// Mitsubishi GX Works2 project: BookEX3_8 Device   PLC: Q13UDV

TYPE DateTime : STRUCT
  Year : INT;
  Month : INT;
  Day : INT;
  WeekDay : INT;
  iHour : INT;
  iMin : INT;
  iSec : INT;
  ms : INT;
END_STRUCT END_TYPE

TYPE Vector : STRUCT
  axisX : REAL;
  axisY : REAL;
  axisZ : REAL;
END_STRUCT END_TYPE

TYPE WordBit : STRUCT
  Data : DWORD;
  Flag : BOOL;
END_STRUCT END_TYPE

// global labels: Global
VAR_GLOBAL
  bVar0 AT M5000 : BOOL;
  abArray0 AT M5010 : ARRAY [0..49] OF BOOL;
  sStr0 AT D5000 : STRING[199];
  sStr1 AT D5100 : STRING[199];
  sStr2 AT D5200 : STRING[199];
  sStr3 AT D5300 : STRING[199];
  sStr4 AT D5400 : STRING[199];
  sStr5 AT D5500 : STRING[199];
  sStr6 AT D5600 : STRING[199];
  sStr7 AT D5700 : STRING[199];
  sStr8 AT D5800 : STRING[199];
  sStr9 AT D5900 : STRING[199];
  iVar0 AT D4500 : INT;
  iVar1 AT D4501 : INT;
  iVar2 AT D4502 : INT;
  iVar3 AT D4503 : INT;
  iVar4 AT D4504 : INT;
  iVar5 AT D4505 : INT;
  iVar6 AT D4506 : INT;
  iVar7 AT D4507 : INT;
  iVar8 AT D4508 : INT;
  iVar9 AT D4509 : INT;
  dVar0 AT D4510 : DINT;
  dVar1 AT D4512 : DINT;
  dVar2 AT D4514 : DINT;
  dVar3 AT D4516 : DINT;
  dVar4 AT D4518 : DINT;
  dVar5 AT D4520 : DINT;
  dVar6 AT D4522 : DINT;
  dVar7 AT D4524 : DINT;
  dVar8 AT D4526 : DINT;
  dVar9 AT D4528 : DINT;
  wVar0 AT D4530 : WORD;
  wVar1 AT D4531 : WORD;
  wVar2 AT D4532 : WORD;
  wVar3 AT D4533 : WORD;
  wVar4 AT D4534 : WORD;
  wVar5 AT D4535 : WORD;
  wVar6 AT D4536 : WORD;
  wVar7 AT D4537 : WORD;
  wVar8 AT D4538 : WORD;
  wVar9 AT D4539 : WORD;
  dwVar0 AT D4540 : DWORD;
  dwVar1 AT D4542 : DWORD;
  dwVar2 AT D4544 : DWORD;
  dwVar3 AT D4546 : DWORD;
  dwVar4 AT D4548 : DWORD;
  dwVar5 AT D4550 : DWORD;
  dwVar6 AT D4552 : DWORD;
  dwVar7 AT D4554 : DWORD;
  dwVar8 AT D4556 : DWORD;
  dwVar9 AT D4558 : DWORD;
  fsVar0 AT D4560 : REAL;
  fsVar1 AT D4562 : REAL;
  fsVar2 AT D4564 : REAL;
  fsVar3 AT D4566 : REAL;
  fsVar4 AT D4568 : REAL;
  fsVar5 AT D4570 : REAL;
  fsVar6 AT D4572 : REAL;
  fsVar7 AT D4574 : REAL;
  fsVar8 AT D4576 : REAL;
  fsVar9 AT D4578 : REAL;
  fdVar0 AT D4580 : LREAL;
  tTime0 AT D4620 : TIME;
  tTime1 AT D4622 : TIME;
  tTime2 AT D4624 : TIME;
  tTime3 AT D4626 : TIME;
  tTime4 AT D4628 : TIME;
  tTime5 AT D4630 : TIME;
  tTime6 AT D4632 : TIME;
  tTime7 AT D4634 : TIME;
  tTime8 AT D4636 : TIME;
  tTime9 AT D4638 : TIME;
  tTime10 AT D4640 : TIME;
  bVar1 AT M5001 : BOOL;
  bVar2 AT M5002 : BOOL;
  bVar3 AT M5003 : BOOL;
  bVar4 AT M5004 : BOOL;
  bVar5 AT M5005 : BOOL;
  bVar6 AT M5006 : BOOL;
  bVar7 AT M5007 : BOOL;
  bVar8 AT M5008 : BOOL;
  bVar9 AT M5009 : BOOL;
  abArray1 AT M5060 : ARRAY [0..49] OF BOOL;
  abArray2 AT M5110 : ARRAY [0..49] OF BOOL;
  abArray3 AT M5160 : ARRAY [0..49] OF BOOL;
  abArray4 AT M5210 : ARRAY [0..49] OF BOOL;
  abArray5 AT M5260 : ARRAY [0..49] OF BOOL;
  abArray6 AT M5310 : ARRAY [0..49] OF BOOL;
  abArray7 AT M5360 : ARRAY [0..49] OF BOOL;
  abArray8 AT M5410 : ARRAY [0..49] OF BOOL;
  abArray9 AT M5460 : ARRAY [0..49] OF BOOL;
  fdVar1 AT D4584 : LREAL;
  fdVar2 AT D4588 : LREAL;
  fdVar3 AT D4592 : LREAL;
  fdVar4 AT D4596 : LREAL;
  fdVar5 AT D4600 : LREAL;
  fdVar6 AT D4604 : LREAL;
  fdVar7 AT D4608 : LREAL;
  fdVar8 AT D4612 : LREAL;
  fdVar9 AT D4616 : LREAL;
  afsPen0 AT D2000 : ARRAY [0..499] OF REAL;
  afsPen1 AT D3000 : ARRAY [0..499] OF REAL;
END_VAR
// user libraries (not included): HMI

PROGRAM 000ConversionLD
VAR
  GetInt : INT;
  NthBit : INT;
  SetInt : INT;
  SetInt2 : INT;
END_VAR
(* structured ladder/FBD written out as ST: instructions are called as NAME(EN, inputs, outputs); _pN, _eN, _tN stand for wires *)
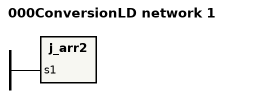
(* network 1 *)
(* element kind 9 j_arr2 <- TRUE *)
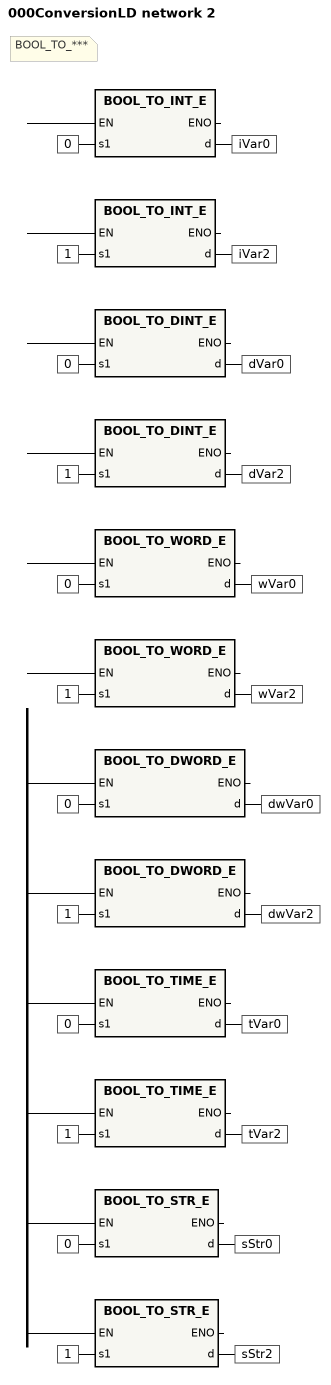
(* network 2 *)
(* BOOL_TO_*** *)
BOOL_TO_INT_E(TRUE, 0, iVar0);
BOOL_TO_INT_E(TRUE, 1, iVar2);
BOOL_TO_DINT_E(TRUE, 0, dVar0);
BOOL_TO_DINT_E(TRUE, 1, dVar2);
BOOL_TO_WORD_E(TRUE, 0, wVar0);
BOOL_TO_WORD_E(TRUE, 1, wVar2);
BOOL_TO_DWORD_E(TRUE, 0, dwVar0);
BOOL_TO_DWORD_E(TRUE, 1, dwVar2);
BOOL_TO_TIME_E(TRUE, 0, tVar0);
BOOL_TO_TIME_E(TRUE, 1, tVar2);
BOOL_TO_STR_E(TRUE, 0, sStr0);
BOOL_TO_STR_E(TRUE, 1, sStr2);
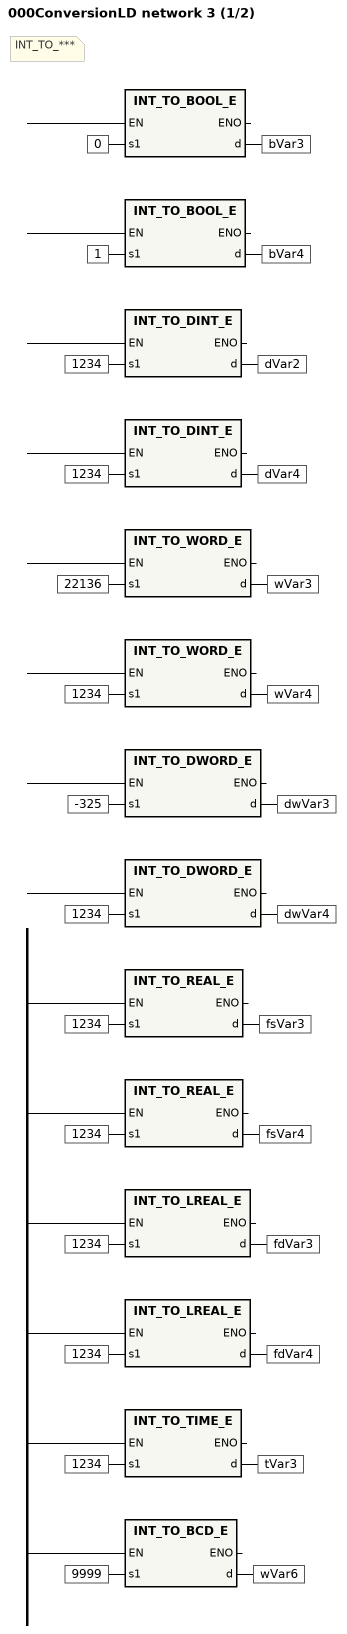
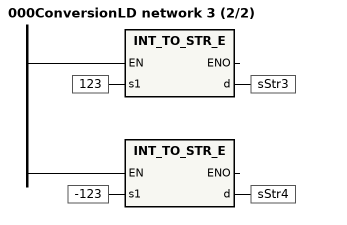
(* network 3 *)
(* INT_TO_*** *)
INT_TO_BOOL_E(TRUE, 0, bVar3);
INT_TO_BOOL_E(TRUE, 1, bVar4);
INT_TO_DINT_E(TRUE, 1234, dVar2);
INT_TO_DINT_E(TRUE, 1234, dVar4);
INT_TO_WORD_E(TRUE, 22136, wVar3);
INT_TO_WORD_E(TRUE, 1234, wVar4);
INT_TO_DWORD_E(TRUE, -325, dwVar3);
INT_TO_DWORD_E(TRUE, 1234, dwVar4);
INT_TO_REAL_E(TRUE, 1234, fsVar3);
INT_TO_REAL_E(TRUE, 1234, fsVar4);
INT_TO_LREAL_E(TRUE, 1234, fdVar3);
INT_TO_LREAL_E(TRUE, 1234, fdVar4);
INT_TO_TIME_E(TRUE, 1234, tVar3);
INT_TO_BCD_E(TRUE, 9999, wVar6);
INT_TO_STR_E(TRUE, 123, sStr3);
INT_TO_STR_E(TRUE, -123, sStr4);
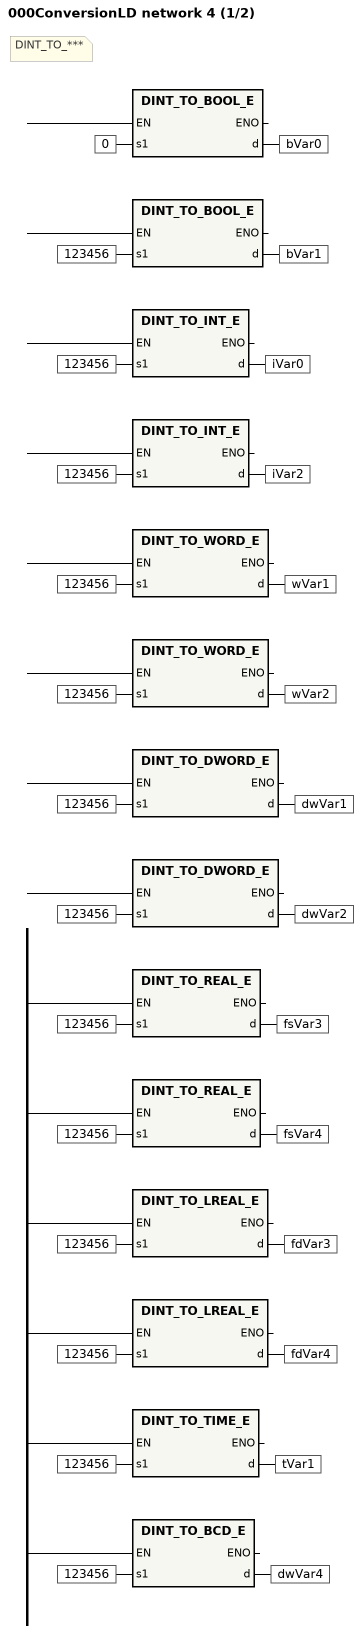
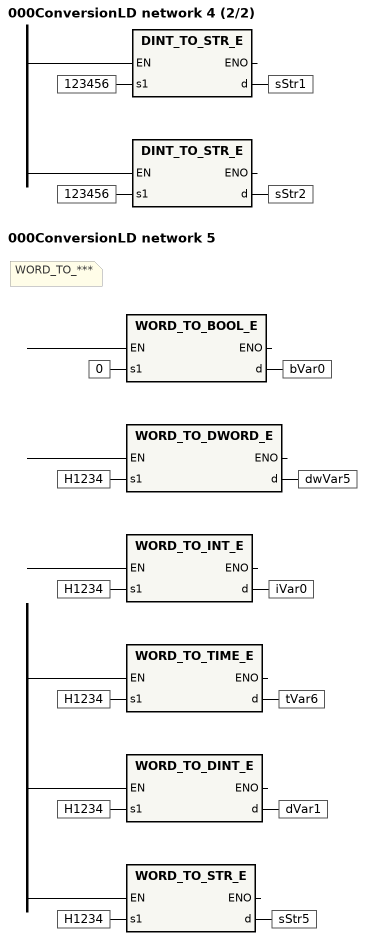
(* network 4 *)
(* DINT_TO_*** *)
DINT_TO_BOOL_E(TRUE, 0, bVar0);
DINT_TO_BOOL_E(TRUE, 123456, bVar1);
DINT_TO_INT_E(TRUE, 123456, iVar0);
DINT_TO_INT_E(TRUE, 123456, iVar2);
DINT_TO_WORD_E(TRUE, 123456, wVar1);
DINT_TO_WORD_E(TRUE, 123456, wVar2);
DINT_TO_DWORD_E(TRUE, 123456, dwVar1);
DINT_TO_DWORD_E(TRUE, 123456, dwVar2);
DINT_TO_REAL_E(TRUE, 123456, fsVar3);
DINT_TO_REAL_E(TRUE, 123456, fsVar4);
DINT_TO_LREAL_E(TRUE, 123456, fdVar3);
DINT_TO_LREAL_E(TRUE, 123456, fdVar4);
DINT_TO_TIME_E(TRUE, 123456, tVar1);
DINT_TO_BCD_E(TRUE, 123456, dwVar4);
DINT_TO_STR_E(TRUE, 123456, sStr1);
DINT_TO_STR_E(TRUE, 123456, sStr2);
(* network 5 *)
(* WORD_TO_*** *)
WORD_TO_BOOL_E(TRUE, 0, bVar0);
WORD_TO_DWORD_E(TRUE, H1234, dwVar5);
WORD_TO_INT_E(TRUE, H1234, iVar0);
WORD_TO_TIME_E(TRUE, H1234, tVar6);
WORD_TO_DINT_E(TRUE, H1234, dVar1);
WORD_TO_STR_E(TRUE, H1234, sStr5);
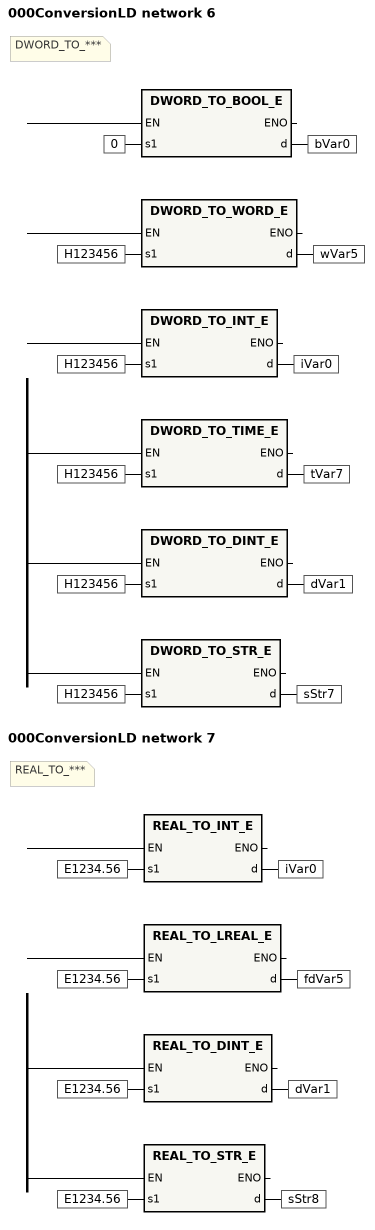
(* network 6 *)
(* DWORD_TO_*** *)
DWORD_TO_BOOL_E(TRUE, 0, bVar0);
DWORD_TO_WORD_E(TRUE, H123456, wVar5);
DWORD_TO_INT_E(TRUE, H123456, iVar0);
DWORD_TO_TIME_E(TRUE, H123456, tVar7);
DWORD_TO_DINT_E(TRUE, H123456, dVar1);
DWORD_TO_STR_E(TRUE, H123456, sStr7);
(* network 7 *)
(* REAL_TO_*** *)
REAL_TO_INT_E(TRUE, E1234.56, iVar0);
REAL_TO_LREAL_E(TRUE, E1234.56, fdVar5);
REAL_TO_DINT_E(TRUE, E1234.56, dVar1);
REAL_TO_STR_E(TRUE, E1234.56, sStr8);
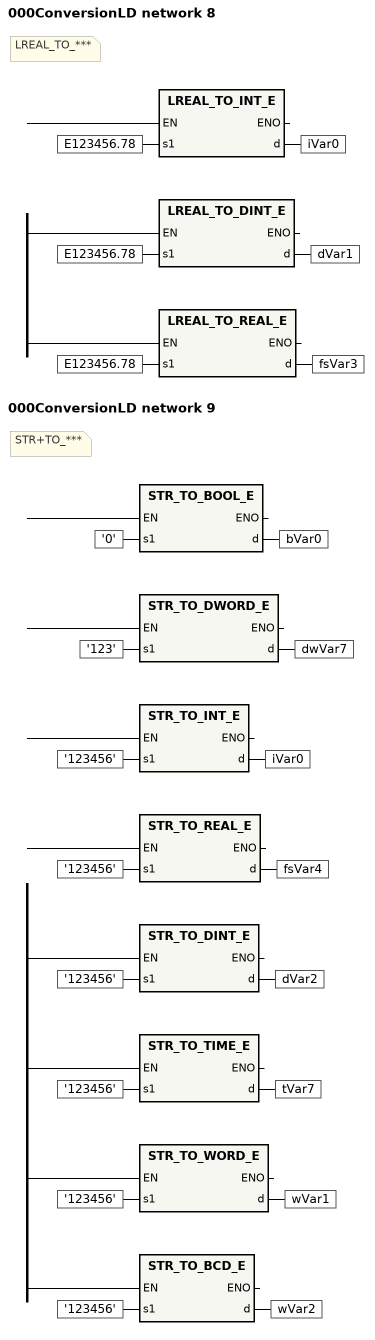
(* network 8 *)
(* LREAL_TO_*** *)
LREAL_TO_INT_E(TRUE, E123456.78, iVar0);
LREAL_TO_DINT_E(TRUE, E123456.78, dVar1);
LREAL_TO_REAL_E(TRUE, E123456.78, fsVar3);
(* network 9 *)
(* STR+TO_*** *)
STR_TO_BOOL_E(TRUE, '0', bVar0);
STR_TO_DWORD_E(TRUE, '123', dwVar7);
STR_TO_INT_E(TRUE, '123456', iVar0);
STR_TO_REAL_E(TRUE, '123456', fsVar4);
STR_TO_DINT_E(TRUE, '123456', dVar2);
STR_TO_TIME_E(TRUE, '123456', tVar7);
STR_TO_WORD_E(TRUE, '123456', wVar1);
STR_TO_BCD_E(TRUE, '123456', wVar2);
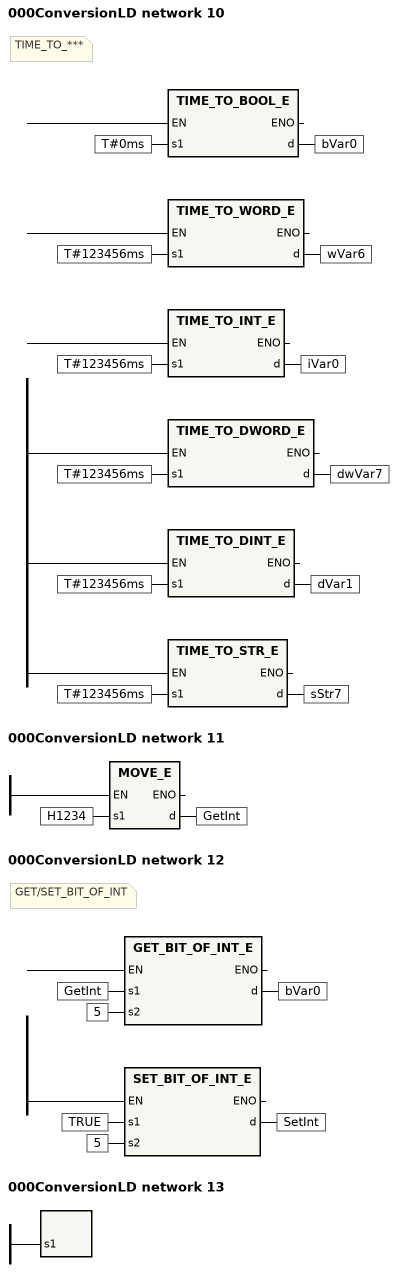
(* network 10 *)
(* TIME_TO_*** *)
TIME_TO_BOOL_E(TRUE, T#0ms, bVar0);
TIME_TO_WORD_E(TRUE, T#123456ms, wVar6);
TIME_TO_INT_E(TRUE, T#123456ms, iVar0);
TIME_TO_DWORD_E(TRUE, T#123456ms, dwVar7);
TIME_TO_DINT_E(TRUE, T#123456ms, dVar1);
TIME_TO_STR_E(TRUE, T#123456ms, sStr7);
(* network 11 Jmp11: *)
MOVE_E(TRUE, H1234, GetInt);
(* network 12 *)
(* GET/SET_BIT_OF_INT *)
GET_BIT_OF_INT_E(TRUE, GetInt, 5, bVar0);
SET_BIT_OF_INT_E(TRUE, TRUE, 5, SetInt);
(* network 13 *)
(* element kind 10  <- TRUE *)
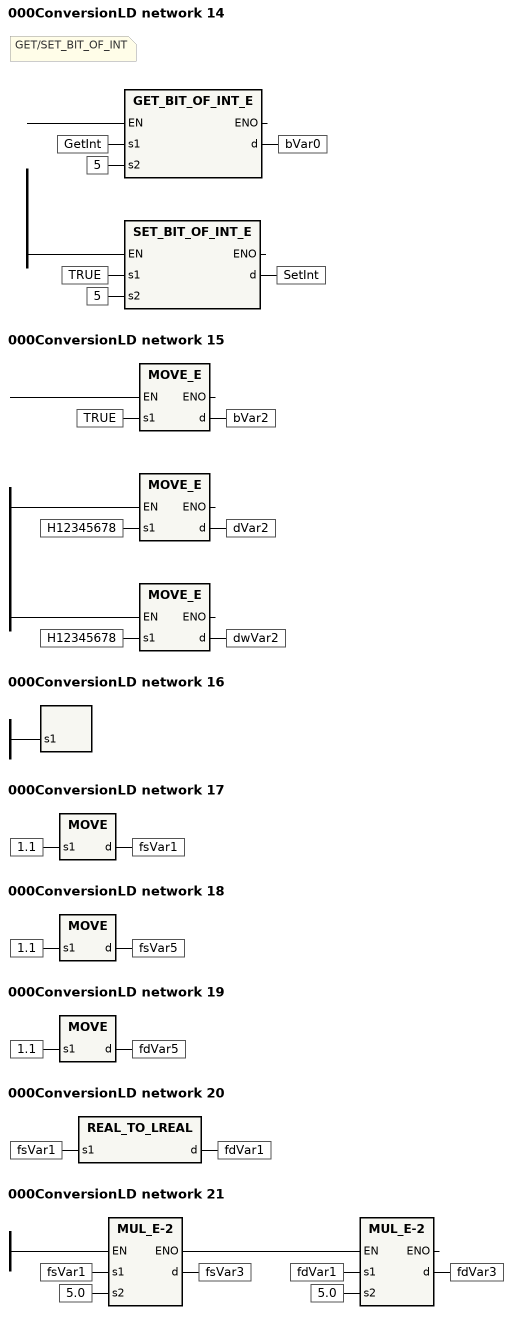
(* network 14 *)
(* GET/SET_BIT_OF_INT *)
GET_BIT_OF_INT_E(TRUE, GetInt, 5, bVar0);
SET_BIT_OF_INT_E(TRUE, TRUE, 5, SetInt);
(* network 15 Jmp15: *)
MOVE_E(TRUE, TRUE, bVar2);
MOVE_E(TRUE, H12345678, dVar2);
MOVE_E(TRUE, H12345678, dwVar2);
(* network 16 *)
(* element kind 10  <- TRUE *)
(* network 17 Jmp20: *)
fsVar1 := MOVE(1.1);
(* network 18 *)
fsVar5 := MOVE(1.1);
(* network 19 *)
fdVar5 := MOVE(1.1);
(* network 20 *)
fdVar1 := REAL_TO_LREAL(fsVar1);
(* network 21 *)
_e1 := MUL_E(TRUE, fsVar1, 5.0, fsVar3);
MUL_E(_e1, fdVar1, 5.0, fdVar3);
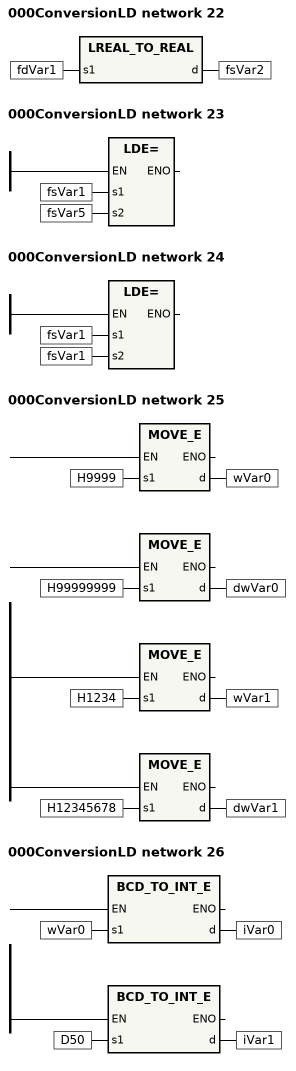
(* network 22 *)
fsVar2 := LREAL_TO_REAL(fdVar1);
(* network 23 *)
LDE=(TRUE, fsVar1, fsVar5);
(* network 24 *)
LDE=(TRUE, fsVar1, fsVar1);
(* network 25 j_bcd: *)
MOVE_E(TRUE, H9999, wVar0);
MOVE_E(TRUE, H99999999, dwVar0);
MOVE_E(TRUE, H1234, wVar1);
MOVE_E(TRUE, H12345678, dwVar1);
(* network 26 *)
BCD_TO_INT_E(TRUE, wVar0, iVar0);
BCD_TO_INT_E(TRUE, D50, iVar1);
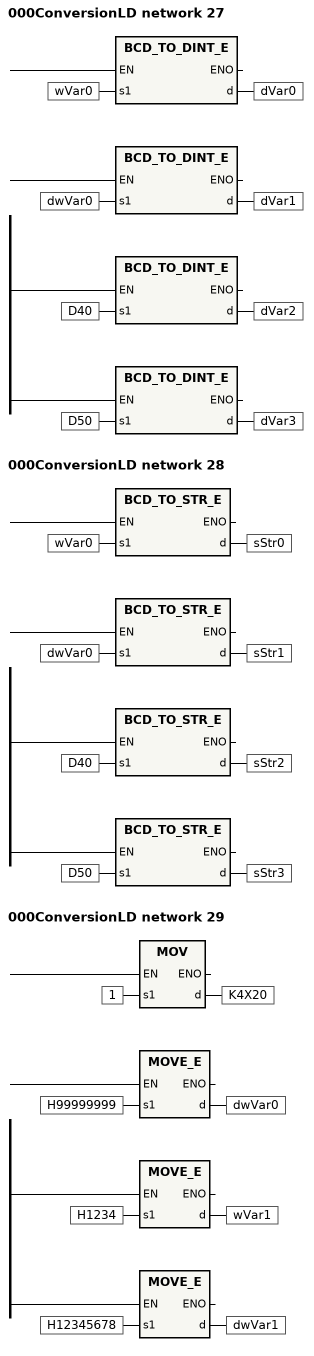
(* network 27 *)
BCD_TO_DINT_E(TRUE, wVar0, dVar0);
BCD_TO_DINT_E(TRUE, dwVar0, dVar1);
BCD_TO_DINT_E(TRUE, D40, dVar2);
BCD_TO_DINT_E(TRUE, D50, dVar3);
(* network 28 *)
BCD_TO_STR_E(TRUE, wVar0, sStr0);
BCD_TO_STR_E(TRUE, dwVar0, sStr1);
BCD_TO_STR_E(TRUE, D40, sStr2);
BCD_TO_STR_E(TRUE, D50, sStr3);
(* network 29 j_deg: *)
MOV(TRUE, 1, K4X20);
MOVE_E(TRUE, H99999999, dwVar0);
MOVE_E(TRUE, H1234, wVar1);
MOVE_E(TRUE, H12345678, dwVar1);
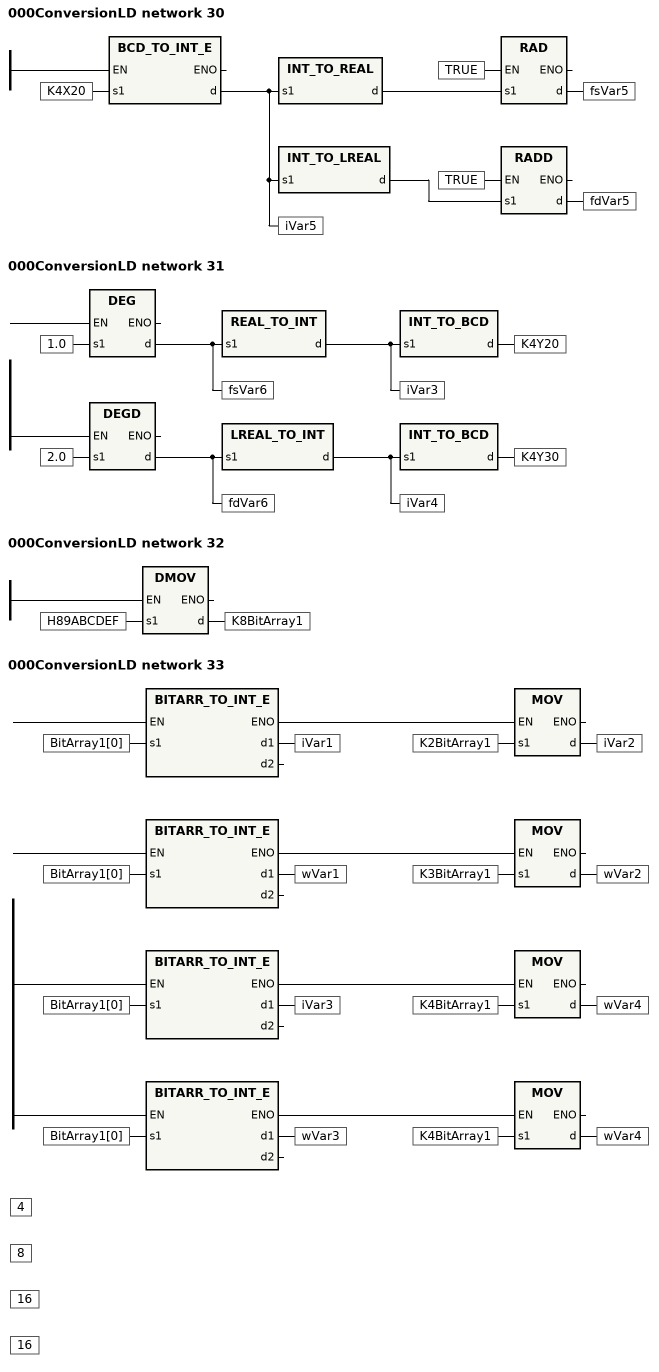
(* network 30 *)
BCD_TO_INT_E(TRUE, K4X20, iVar5);
RAD(TRUE, INT_TO_REAL(iVar5), fsVar5);
RADD(TRUE, INT_TO_LREAL(iVar5), fdVar5);
(* network 31 *)
DEG(TRUE, 1.0, fsVar6);
_p1 := REAL_TO_INT(fsVar6);
iVar3 := _p1;
K4Y20 := INT_TO_BCD(_p1);
DEGD(TRUE, 2.0, fdVar6);
_p2 := LREAL_TO_INT(fdVar6);
iVar4 := _p2;
K4Y30 := INT_TO_BCD(_p2);
(* network 32 j_arr: *)
DMOV(TRUE, H89ABCDEF, K8BitArray1);
(* network 33 *)
_e1 := BITARR_TO_INT_E(TRUE, BitArray1[0], iVar1, _open);
MOV(_e1, K2BitArray1, iVar2);
_e2 := BITARR_TO_INT_E(TRUE, BitArray1[0], wVar1, _open);
MOV(_e2, K3BitArray1, wVar2);
_e3 := BITARR_TO_INT_E(TRUE, BitArray1[0], iVar3, _open);
MOV(_e3, K4BitArray1, wVar4);
_e4 := BITARR_TO_INT_E(TRUE, BitArray1[0], wVar3, _open);
MOV(_e4, K4BitArray1, wVar4);
(* not connected to any output: 4, 8, 16, 16 *)
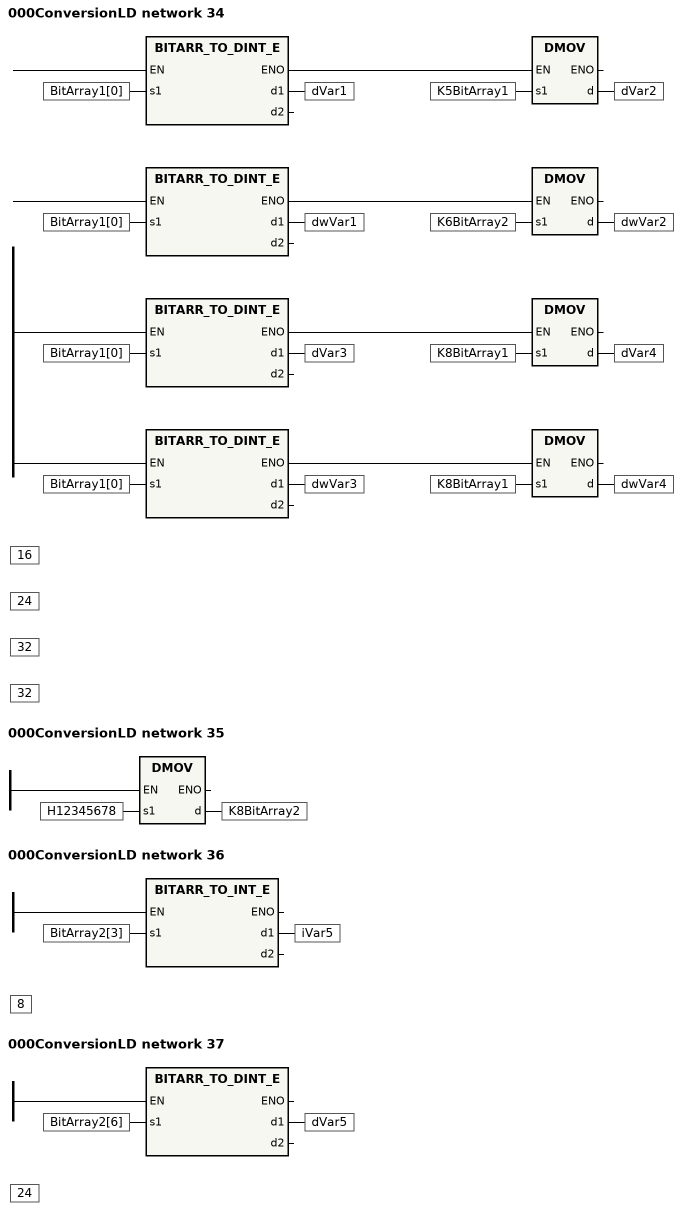
(* network 34 *)
_e1 := BITARR_TO_DINT_E(TRUE, BitArray1[0], dVar1, _open);
DMOV(_e1, K5BitArray1, dVar2);
_e2 := BITARR_TO_DINT_E(TRUE, BitArray1[0], dwVar1, _open);
DMOV(_e2, K6BitArray2, dwVar2);
_e3 := BITARR_TO_DINT_E(TRUE, BitArray1[0], dVar3, _open);
DMOV(_e3, K8BitArray1, dVar4);
_e4 := BITARR_TO_DINT_E(TRUE, BitArray1[0], dwVar3, _open);
DMOV(_e4, K8BitArray1, dwVar4);
(* not connected to any output: 16, 24, 32, 32 *)
(* network 35 *)
DMOV(TRUE, H12345678, K8BitArray2);
(* network 36 *)
BITARR_TO_INT_E(TRUE, BitArray2[3], iVar5, _open);
(* not connected to any output: 8 *)
(* network 37 *)
BITARR_TO_DINT_E(TRUE, BitArray2[6], dVar5, _open);
(* not connected to any output: 24 *)
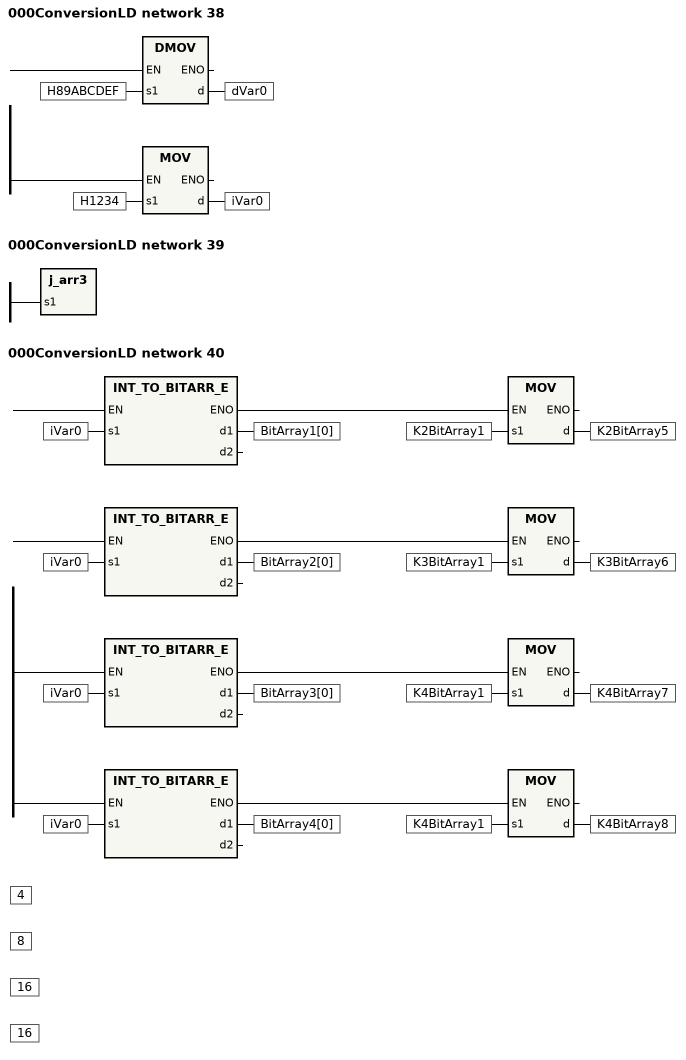
(* network 38 j_arr2: *)
DMOV(TRUE, H89ABCDEF, dVar0);
MOV(TRUE, H1234, iVar0);
(* network 39 *)
(* element kind 9 j_arr3 <- TRUE *)
(* network 40 *)
_e1 := INT_TO_BITARR_E(TRUE, iVar0, BitArray1[0], _open);
MOV(_e1, K2BitArray1, K2BitArray5);
_e2 := INT_TO_BITARR_E(TRUE, iVar0, BitArray2[0], _open);
MOV(_e2, K3BitArray1, K3BitArray6);
_e3 := INT_TO_BITARR_E(TRUE, iVar0, BitArray3[0], _open);
MOV(_e3, K4BitArray1, K4BitArray7);
_e4 := INT_TO_BITARR_E(TRUE, iVar0, BitArray4[0], _open);
MOV(_e4, K4BitArray1, K4BitArray8);
(* not connected to any output: 4, 8, 16, 16 *)
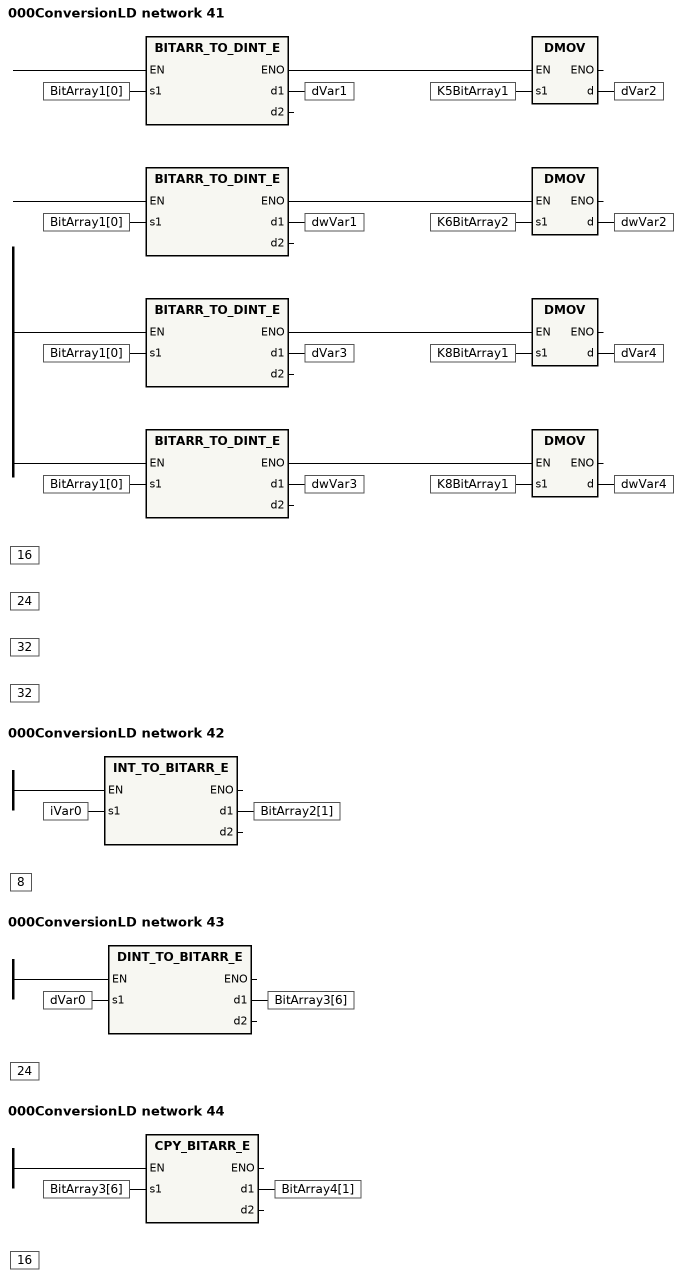
(* network 41 *)
_e1 := BITARR_TO_DINT_E(TRUE, BitArray1[0], dVar1, _open);
DMOV(_e1, K5BitArray1, dVar2);
_e2 := BITARR_TO_DINT_E(TRUE, BitArray1[0], dwVar1, _open);
DMOV(_e2, K6BitArray2, dwVar2);
_e3 := BITARR_TO_DINT_E(TRUE, BitArray1[0], dVar3, _open);
DMOV(_e3, K8BitArray1, dVar4);
_e4 := BITARR_TO_DINT_E(TRUE, BitArray1[0], dwVar3, _open);
DMOV(_e4, K8BitArray1, dwVar4);
(* not connected to any output: 16, 24, 32, 32 *)
(* network 42 j_arr3: *)
INT_TO_BITARR_E(TRUE, iVar0, BitArray2[1], _open);
(* not connected to any output: 8 *)
(* network 43 *)
DINT_TO_BITARR_E(TRUE, dVar0, BitArray3[6], _open);
(* not connected to any output: 24 *)
(* network 44 *)
CPY_BITARR_E(TRUE, BitArray3[6], BitArray4[1], _open);
(* not connected to any output: 16 *)
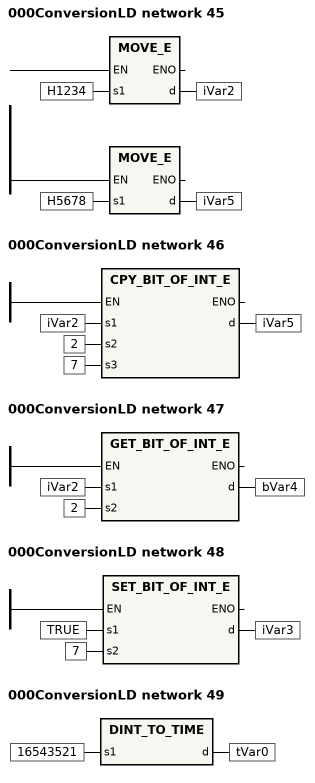
(* network 45 *)
MOVE_E(TRUE, H1234, iVar2);
MOVE_E(TRUE, H5678, iVar5);
(* network 46 *)
CPY_BIT_OF_INT_E(TRUE, iVar2, 2, 7, iVar5);
(* network 47 *)
GET_BIT_OF_INT_E(TRUE, iVar2, 2, bVar4);
(* network 48 *)
SET_BIT_OF_INT_E(TRUE, TRUE, 7, iVar3);
(* network 49 *)
tVar0 := DINT_TO_TIME(16543521);
END_PROGRAM

PROGRAM 000DataType(FBD)
VAR
  aClock : ARRAY [0..6] OF INT;
  awStatus : ARRAY [0..9] OF WORD;
  asName : ARRAY [0..4] OF STRING[32] := [5('')];
  atDelay : ARRAY [0..4] OF TIME := [5(T#0s)];
  asStr : STRING[32];
  Word2Bool2_1 : Word2Bit;
  Word2Bool_1 : Word2Bit;
END_VAR
(* structured ladder/FBD written out as ST: instructions are called as NAME(EN, inputs, outputs); _pN, _eN, _tN stand for wires *)
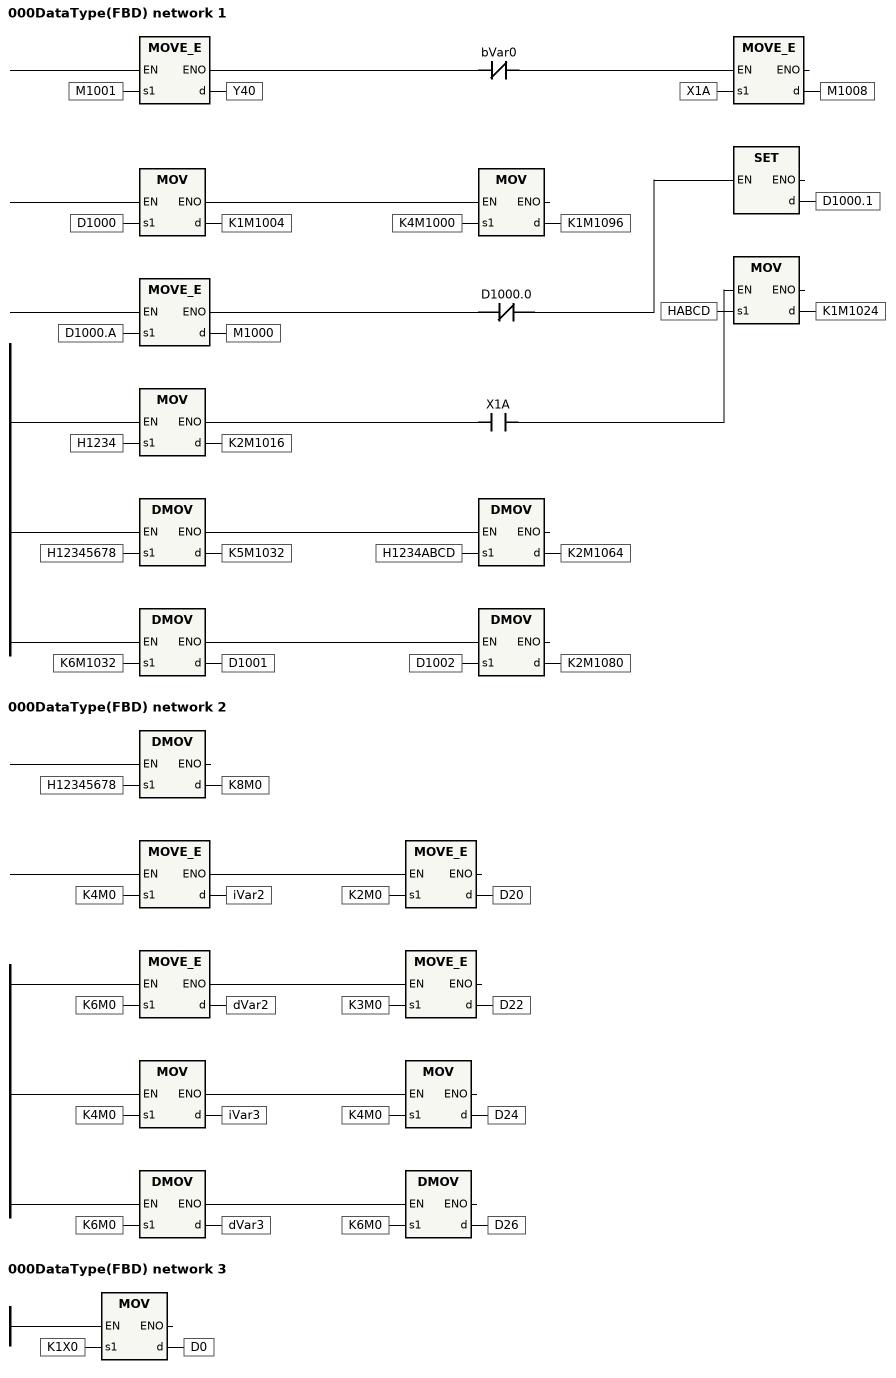
(* network 1 *)
_e1 := MOVE_E(TRUE, M1001, Y40);
MOVE_E(_e1 AND NOT bVar0, X1A, M1008);
_e2 := MOVE_E(TRUE, D1000.A, M1000);
SET(_e2 AND NOT D1000.0, D1000.1);
_e3 := MOV(TRUE, H1234, K2M1016);
MOV(_e3 AND X1A, HABCD, K1M1024);
_e4 := MOV(TRUE, D1000, K1M1004);
MOV(_e4, K4M1000, K1M1096);
_e5 := DMOV(TRUE, H12345678, K5M1032);
DMOV(_e5, H1234ABCD, K2M1064);
_e6 := DMOV(TRUE, K6M1032, D1001);
DMOV(_e6, D1002, K2M1080);
(* network 2 *)
DMOV(TRUE, H12345678, K8M0);
_e1 := MOVE_E(TRUE, K4M0, iVar2);
MOVE_E(_e1, K2M0, D20);
_e2 := MOVE_E(TRUE, K6M0, dVar2);
MOVE_E(_e2, K3M0, D22);
_e3 := MOV(TRUE, K4M0, iVar3);
MOV(_e3, K4M0, D24);
_e4 := DMOV(TRUE, K6M0, dVar3);
DMOV(_e4, K6M0, D26);
(* network 3 *)
MOV(TRUE, K1X0, D0);
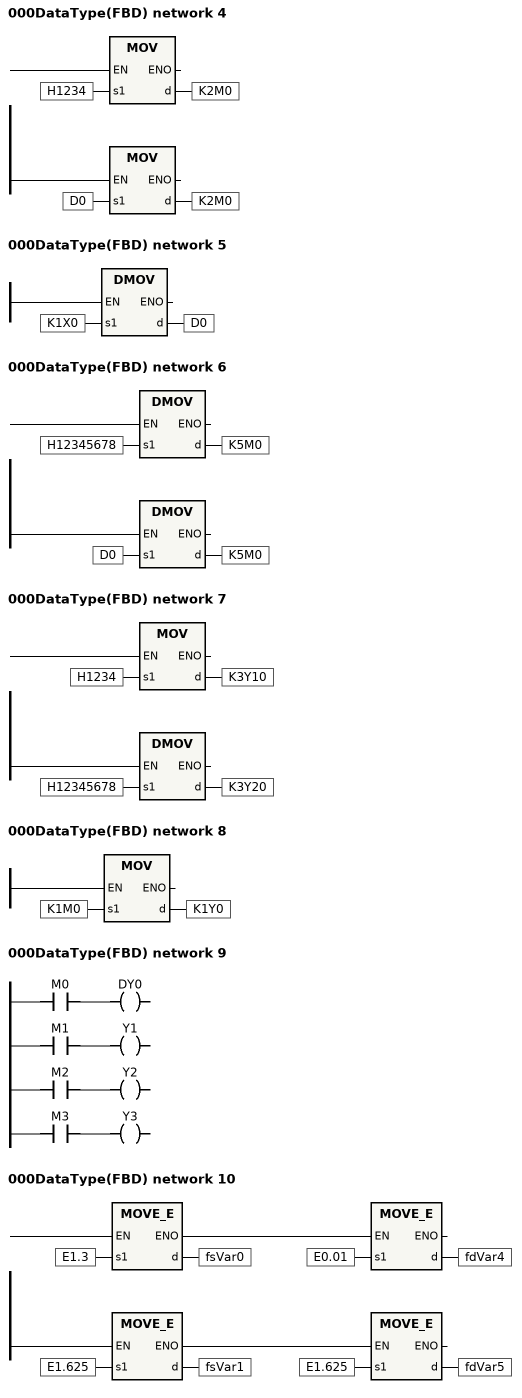
(* network 4 *)
MOV(TRUE, H1234, K2M0);
MOV(TRUE, D0, K2M0);
(* network 5 *)
DMOV(TRUE, K1X0, D0);
(* network 6 *)
DMOV(TRUE, H12345678, K5M0);
DMOV(TRUE, D0, K5M0);
(* network 7 *)
MOV(TRUE, H1234, K3Y10);
DMOV(TRUE, H12345678, K3Y20);
(* network 8 *)
MOV(TRUE, K1M0, K1Y0);
(* network 9 *)
DY0 := M0;
Y1 := M1;
Y2 := M2;
Y3 := M3;
(* network 10 *)
_e1 := MOVE_E(TRUE, E1.3, fsVar0);
MOVE_E(_e1, E0.01, fdVar4);
_e2 := MOVE_E(TRUE, E1.625, fsVar1);
MOVE_E(_e2, E1.625, fdVar5);
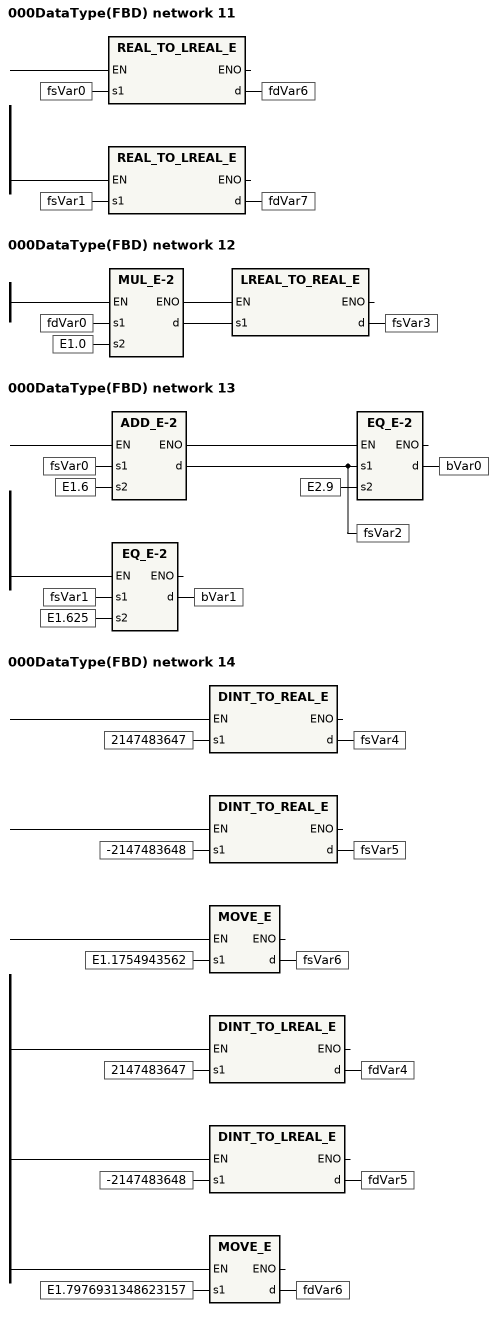
(* network 11 *)
REAL_TO_LREAL_E(TRUE, fsVar0, fdVar6);
REAL_TO_LREAL_E(TRUE, fsVar1, fdVar7);
(* network 12 *)
_e2 := MUL_E(TRUE, fdVar0, E1.0, _t1);
LREAL_TO_REAL_E(_e2, _t1, fsVar3);
(* network 13 *)
_e1 := ADD_E(TRUE, fsVar0, E1.6, fsVar2);
EQ_E(_e1, fsVar2, E2.9, bVar0);
EQ_E(TRUE, fsVar1, E1.625, bVar1);
(* network 14 *)
DINT_TO_REAL_E(TRUE, 2147483647, fsVar4);
DINT_TO_REAL_E(TRUE, -2147483648, fsVar5);
MOVE_E(TRUE, E1.1754943562, fsVar6);
DINT_TO_LREAL_E(TRUE, 2147483647, fdVar4);
DINT_TO_LREAL_E(TRUE, -2147483648, fdVar5);
MOVE_E(TRUE, E1.7976931348623157, fdVar6);
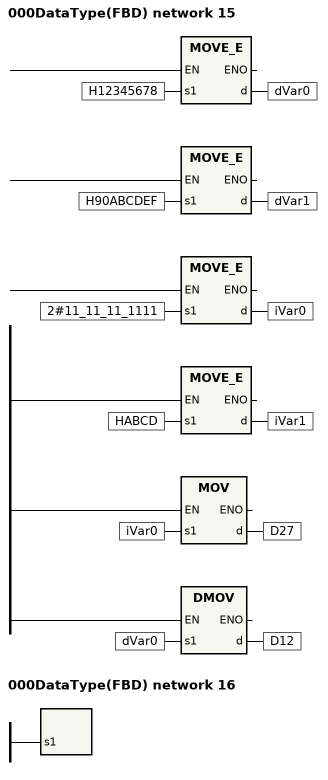
(* network 15 *)
MOVE_E(TRUE, H12345678, dVar0);
MOVE_E(TRUE, H90ABCDEF, dVar1);
MOVE_E(TRUE, 2#11_11_11_1111, iVar0);
MOVE_E(TRUE, HABCD, iVar1);
MOV(TRUE, iVar0, D27);
DMOV(TRUE, dVar0, D12);
(* network 16 *)
(* element kind 10  <- TRUE *)
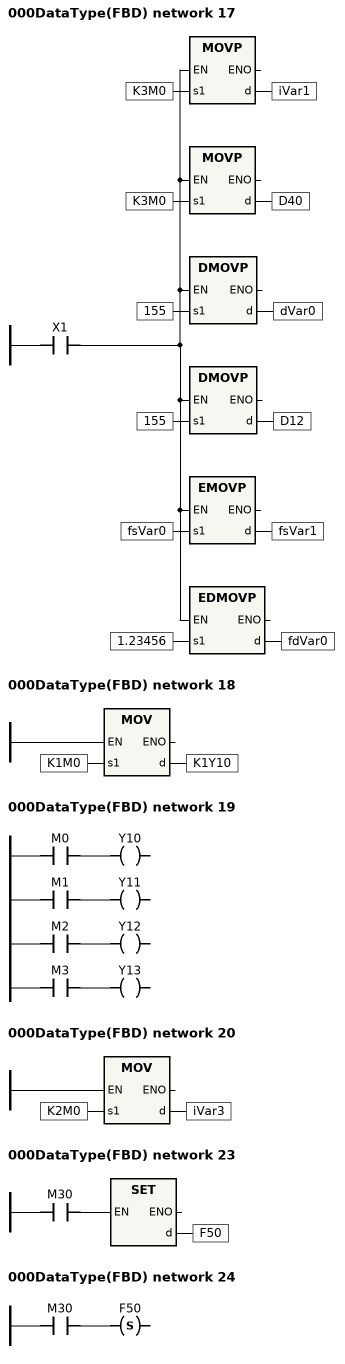
(* network 17 jmp_mov: *)
MOVP(X1, K3M0, iVar1);
MOVP(X1, K3M0, D40);
DMOVP(X1, 155, dVar0);
DMOVP(X1, 155, D12);
EMOVP(X1, fsVar0, fsVar1);
EDMOVP(X1, 1.23456, fdVar0);
(* network 18 *)
MOV(TRUE, K1M0, K1Y10);
(* network 19 *)
Y10 := M0;
Y11 := M1;
Y12 := M2;
Y13 := M3;
(* network 20 *)
MOV(TRUE, K2M0, iVar3);
(* network 23 j_mov3: *)
SET(M30, F50);
(* network 24 *)
SET(M30, F50);
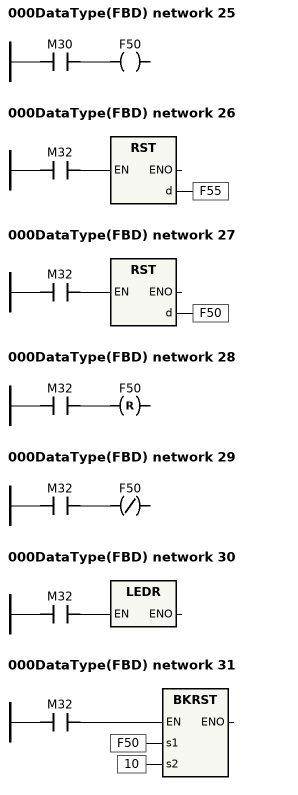
(* network 25 *)
F50 := M30;
(* network 26 *)
RST(M32, F55);
(* network 27 *)
RST(M32, F50);
(* network 28 *)
RST(M32, F50);
(* network 29 *)
F50 := NOT M32;
(* network 30 *)
LEDR(M32);
(* network 31 *)
BKRST(M32, F50, 10);
END_PROGRAM

PROGRAM ADRTest
(* structured ladder/FBD written out as ST: instructions are called as NAME(EN, inputs, outputs); _pN, _eN, _tN stand for wires *)
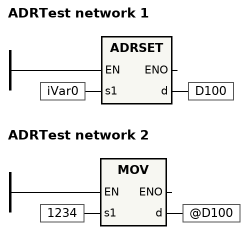
(* network 1 *)
ADRSET(TRUE, iVar0, D100);
(* network 2 *)
MOV(TRUE, 1234, @D100);
END_PROGRAM

PROGRAM ExDevice
VAR
  bMreg : BOOL;
  Mov4INT_1 : Mov4INT;
  Mov8INT_1 : Mov8INT;
END_VAR
(* structured ladder/FBD written out as ST: instructions are called as NAME(EN, inputs, outputs); _pN, _eN, _tN stand for wires *)
